Staubli VAL3: setActive.pgx

public program setActive(bool x_bActive, string x_sItem)
  local num l_nSize
begin
  // check if is active
  saveInOut:dInput[x_sItem].bActive=x_bActive
end
